                | elif(var_2 == "34"):
                |   movej(p[-0.62575,-0.525,0.05075,2.230,2.215,0])
                | elif(var_2 == "35"):
                |   movej(p[-0.72575,0.525,0.05075,2.230,2.215,0])
                | elif(var_2 == "36"):
                |   movej(p[-0.72575,0.350,0.05075,2.230,2.215,0])
                | elif(var_2 == "37"):
                |   movej(p[-0.72575,0.175,0.05075,2.230,2.215,0])
                | elif(var_2 == "38"):
                |   movej(p[-0.72575,0,0.05075,2.230,2.215,0])
                | elif(var_2 == "39"):
                |   movej(p[-0.72575,-0.175,0.05075,2.230,2.215,0])
                | elif(var_2 == "40"):
                |   movej(p[-0.72575,-0.350,0.05075,2.230,2.215,0])
                | elif(var_2 == "41"):
                |   movej(p[-0.72575,-0.525,0.05075,2.230,2.215,0])
                | elif(var_2 == "42"):
                |   movej(p[-0.82575,0.525,0.05075,2.230,2.215,0])
                | elif(var_2 == "43"):
                |   movej(p[-0.82575,0.350,0.05075,2.230,2.215,0])
                | elif(var_2 == "44"):
                |   movej(p[-0.82575,0.175,0.05075,2.230,2.215,0])
                | elif(var_2 == "45"):
                |   movej(p[-0.82575,0,0.05075,2.230,2.215,0])
                | elif(var_2 == "46"):
                |   movej(p[-0.82575,-0.175,0.05075,2.230,2.215,0])
                | elif(var_2 == "47"):
                |   movej(p[-0.82575,-0.350,0.05075,2.230,2.215,0])
                | elif(var_2 == "48"):
                |   movej(p[-0.82575,-0.525,0.05075,2.230,2.215,0])
                | elif(var_2 == "49"):
                |   movej(p[-0.92575,0.525,0.05075,2.230,2.215,0])
                | elif(var_2 == "50"):
                |   movej(p[-0.92575,0.350,0.05075,2.230,2.215,0])
                | elif(var_2 == "51"):
                |   movej(p[-0.92575,0.175,0.05075,2.230,2.215,0])
                | elif(var_2 == "52"):
                |   movej(p[-0.92575,0,0.05075,2.230,2.215,0])
                | elif(var_2 == "53"):
                |   movej(p[-0.92575,-0.175,0.05075,2.230,2.215,0])
                | elif(var_2 == "54"):
                |   movej(p[-0.92575,-0.350,0.05075,2.230,2.215,0])
                | elif(var_2 == "55"):
                |   movej(p[-0.92575,-0.525,0.05075,2.230,2.215,0])
                | elif(var_2 == "56"):
                |   movej(p[-1.02575,0.525,0.05075,2.230,2.215,0])
                | elif(var_2 == "57"):
                |   movej(p[-1.02575,0.350,0.05075,2.230,2.215,0])
                | elif(var_2 == "58"):
                |   movej(p[-1.02575,0.175,0.05075,2.230,2.215,0])
                | elif(var_2 == "59"):
                |   movej(p[-1.02575,0,0.05075,2.230,2.215,0])
                | elif(var_2 == "60"):
                |   movej(p[-1.02575,-0.175,0.05075,2.230,2.215,0])
                | elif(var_2 == "61"):
                |   movej(p[-1.02575,-0.350,0.05075,2.230,2.215,0])
                | elif(var_2 == "62"):
                |   movej(p[-1.02575,-0.525,0.05075,2.230,2.215,0])
                | elif(var_2 == "71"):
                |   movej(p[-0.600,-1.050,-0.220,0,3.14,0])
                | elif(var_2 == "72"):
                |   movej(p[-0.380,-1.050,-0.220,0,3.14,0])
                | elif(var_2 == "73"):
                |   movej(p[-0.160,-1.050,-0.220,0,3.14,0])
                | elif(var_2 == "74"):
                |   movej(p[0.060,-1.050,-0.220,0,3.14,0])
                | elif(var_2 == "75"):
                |   movej(p[0.280,-1.050,-0.220,0,3.14,0])
                | elif(var_2 == "76"):
                |   movej(p[0.500,-1.050,-0.220,0,3.14,0])
                | end
              Wait Sleep waitTime=0.5
              top_pos1 := get_actual_tcp_pose()
              Script: top_pos1[2] = top_pos1[2]-0.15
              MoveJ speed 60 deg/s, acceleration 80 deg/s^2 (useActiveTCP=true)
                Waypoint Waypoint (Variable): variable=top_pos1
              URCap Vacuum (Robotiq_Grippers, Robotiq Inc.) dataModel(Vacuum.Command.Action=1, Vacuum.Command.PumpAutoCloseDelayInMilliseconds=3000, Vacuum.Command.ShutOffDistance=5.0)
              Wait Sleep waitTime=0.5
              Script: var_4 =  False
              MoveJ speed 60 deg/s, acceleration 80 deg/s^2 (useActiveTCP=true)
                Waypoint place_pos: motionParameters(blendRadius=0.05); TCP in base x=-418.268 y=159.557 z=391.133 mm, rx=-2.2681 ry=-2.171 rz=-0.0004 rad; joints [-180.311, -63.896, -116.331, -89.8, 89.467, 2.625] deg; flange x=-418.043 y=159.256 z=582.133 mm, rx=-2.2681 ry=-2.171 rz=-0.0004 rad
            Else 
              MoveJ speed 60 deg/s, acceleration 80 deg/s^2 (useActiveTCP=true)
                Waypoint place_pos: motionParameters(blendRadius=0.05); TCP in base x=-418.268 y=159.557 z=391.133 mm, rx=-2.2681 ry=-2.171 rz=-0.0004 rad; joints [-180.311, -63.896, -116.331, -89.8, 89.467, 2.625] deg; flange x=-418.043 y=159.256 z=582.133 mm, rx=-2.2681 ry=-2.171 rz=-0.0004 rad
          Wait Sleep waitTime=0.5
          MoveJ speed 60 deg/s, acceleration 80 deg/s^2 (useActiveTCP=true)
            Waypoint Waypoint_10: TCP in base x=-0.074 y=-449.982 z=400.013 mm, rx=2.1808 ry=-2.261 rz=0.0021 rad; joints [-69.631, -64.171, -115.295, -90.553, 89.57, -67.123] deg; flange x=-0.215 y=-449.768 z=591.013 mm, rx=2.1808 ry=-2.261 rz=0.0021 rad
          Folder T12
            If var_3 =="201"
              MoveJ speed 60 deg/s, acceleration 80 deg/s^2 (useActiveTCP=true)
                Waypoint Waypoint_7: TCP in base x=69.993 y=-340.039 z=51.5 mm, rx=2.1806 ry=-2.2612 rz=0.0018 rad; joints [-50.861, -64.539, -152.673, -52.818, 89.717, -48.758] deg; flange x=69.876 y=-339.852 z=242.5 mm, rx=2.1806 ry=-2.2612 rz=0.0018 rad
              Script: var_4 =  True
            ElseIf var_3 == "202"
              MoveJ speed 60 deg/s, acceleration 80 deg/s^2 (useActiveTCP=true)
                Waypoint Waypoint_8: TCP in base x=-65.595 y=-340.045 z=51.514 mm, rx=2.1805 ry=-2.2613 rz=0.0019 rad; joints [-73.362, -64.391, -152.734, -52.902, 89.747, -71.257] deg; flange x=-65.727 y=-339.849 z=242.514 mm, rx=2.1805 ry=-2.2613 rz=0.0019 rad
              Script: var_4 =  True
            ElseIf var_3 =="203"
              MoveJ speed 60 deg/s, acceleration 80 deg/s^2 (useActiveTCP=true)
                Waypoint Waypoint_9: TCP in base x=-194.737 y=-340.099 z=51.532 mm, rx=2.1807 ry=-2.2612 rz=0.0019 rad; joints [-95.738, -71.977, -149.014, -49.049, 89.723, -93.648] deg; flange x=-194.869 y=-339.905 z=242.532 mm, rx=2.1807 ry=-2.2612 rz=0.0019 rad
              Script: var_4 =  True
            ElseIf var_3 == "204"
              Script: var_4 =  False
            If var_4 ==  True
              URCap Find Surface (Robotiq_Copilot, Robotiq Inc.) dataModel(NodeInitializedKey=true, WaitForSteadyWrenchOptionKey=false, ls_force=10.0, ZeroSensorBeforeKey=true, ls_distance=500.0, ls_speed=50.0, ls_direction=Z-, FindSurfaceFeatureKey=0, ls_if_distance=false, ls_if_force=false); state(isChildrenLocked=true)
                'Add Stop conditions from the Find Surface node'
              URCap Vacuum (Robotiq_Grippers, Robotiq Inc.) dataModel(Vacuum.Command.GripMode=Manual, Vacuum.Command.MinVacuumInPercent=70.0, Vacuum.Command.MaxVacuumInPercent=90.0, Vacuum.Command.Action=0, Vacuum.Command.PumpAutoCloseDelayInMilliseconds=3000, Vacuum.Command.ShutOffDistance=5.0)
              Wait Sleep waitTime=0.5
              top_pos2 := get_actual_tcp_pose()
              Script: top_pos2[2] = top_pos2[2]+0.01
              MoveJ speed 60 deg/s, acceleration 80 deg/s^2 (useActiveTCP=true)
                Waypoint Waypoint (Variable): variable=top_pos2
                Waypoint Waypoint_10: TCP in base x=-0.074 y=-449.982 z=400.013 mm, rx=2.1808 ry=-2.261 rz=0.0021 rad; joints [-69.631, -64.171, -115.295, -90.553, 89.57, -67.123] deg; flange x=-0.215 y=-449.768 z=591.013 mm, rx=2.1808 ry=-2.261 rz=0.0021 rad
              Wait Sleep waitTime=0.5
              MoveJ speed 60 deg/s, acceleration 80 deg/s^2 (useActiveTCP=true)
                Waypoint place_pos: motionParameters(blendRadius=0.05); TCP in base x=-418.268 y=159.557 z=391.133 mm, rx=-2.2681 ry=-2.171 rz=-0.0004 rad; joints [-180.311, -63.896, -116.331, -89.8, 89.467, 2.625] deg; flange x=-418.043 y=159.256 z=582.133 mm, rx=-2.2681 ry=-2.171 rz=-0.0004 rad
              Wait Sleep waitTime=0.5
              Script file /programs/new dir/place3.script
                | (same text as the earlier copy of this file)
              Wait Sleep waitTime=0.5
              top_pos1 := get_actual_tcp_pose()
              Script: top_pos1[2] = top_pos1[2]-0.15
              MoveJ speed 60 deg/s, acceleration 80 deg/s^2 (useActiveTCP=true)
                Waypoint Waypoint (Variable): variable=top_pos1
              URCap Vacuum (Robotiq_Grippers, Robotiq Inc.) dataModel(Vacuum.Command.Action=1, Vacuum.Command.PumpAutoCloseDelayInMilliseconds=3000, Vacuum.Command.ShutOffDistance=5.0)
              Wait Sleep waitTime=0.5
              Script: var_4 =  False
              MoveJ speed 60 deg/s, acceleration 80 deg/s^2 (useActiveTCP=true)
                Waypoint place_pos: motionParameters(blendRadius=0.05); TCP in base x=-418.268 y=159.557 z=391.133 mm, rx=-2.2681 ry=-2.171 rz=-0.0004 rad; joints [-180.311, -63.896, -116.331, -89.8, 89.467, 2.625] deg; flange x=-418.043 y=159.256 z=582.133 mm, rx=-2.2681 ry=-2.171 rz=-0.0004 rad
            Else 
              MoveJ speed 60 deg/s, acceleration 80 deg/s^2 (useActiveTCP=true)
                Waypoint place_pos: motionParameters(blendRadius=0.05); TCP in base x=-418.268 y=159.557 z=391.133 mm, rx=-2.2681 ry=-2.171 rz=-0.0004 rad; joints [-180.311, -63.896, -116.331, -89.8, 89.467, 2.625] deg; flange x=-418.043 y=159.256 z=582.133 mm, rx=-2.2681 ry=-2.171 rz=-0.0004 rad
          MoveJ speed 60 deg/s, acceleration 80 deg/s^2 (useActiveTCP=true)
            Waypoint Waypoint_10: TCP in base x=-0.074 y=-449.982 z=400.013 mm, rx=2.1808 ry=-2.261 rz=0.0021 rad; joints [-69.631, -64.171, -115.295, -90.553, 89.57, -67.123] deg; flange x=-0.215 y=-449.768 z=591.013 mm, rx=2.1808 ry=-2.261 rz=0.0021 rad
          Script: socket_send_string("top_placed")
          Wait Sleep waitTime=0.5
          If var_2 == "5"
            MoveJ speed 60 deg/s, acceleration 80 deg/s^2 (useActiveTCP=true)
              Waypoint place_pos: motionParameters(blendRadius=0.05); TCP in base x=-418.268 y=159.557 z=391.133 mm, rx=-2.2681 ry=-2.171 rz=-0.0004 rad; joints [-180.311, -63.896, -116.331, -89.8, 89.467, 2.625] deg; flange x=-418.043 y=159.256 z=582.133 mm, rx=-2.2681 ry=-2.171 rz=-0.0004 rad
            Script: break
      Folder Push
        var_5 := 0
        Wait Sleep waitTime=0.5
        If var_5 == 0
          MoveJ speed 60 deg/s, acceleration 80 deg/s^2 (useActiveTCP=true)
            Waypoint Waypoint_12: TCP in base x=-158.301 y=504.125 z=400.028 mm, rx=-0.0124 ry=-3.1401 rz=0.0022 rad; joints [-235.391, -72.645, -110.118, -87.346, 89.583, -144.51] deg; flange x=-158.011 y=504.388 z=591.028 mm, rx=-0.0124 ry=-3.1401 rz=0.0022 rad
            Waypoint Waypoint_15: TCP in base x=-170.086 y=486.92 z=61.096 mm, rx=-0.0304 ry=-3.1398 rz=0.0019 rad; joints [-232.86, -86.331, -137.199, -46.56, 89.659, -141.738] deg; flange x=-169.765 y=487.153 z=252.096 mm, rx=-0.0304 ry=-3.1398 rz=0.0019 rad
          Wait Sleep waitTime=0.5
          MoveL speed 250 mm/s, acceleration 1200 mm/s^2 (useActiveTCP=true) feature=Base
            Waypoint Waypoint_13: TCP in base x=-1165 y=500.206 z=60.955 mm, rx=-0.0455 ry=-3.1398 rz=0.002 rad; joints [-195.929, -158.624, -21.708, -89.701, 88.788, -104.245] deg; flange x=-1164.721 y=500.444 z=251.955 mm, rx=-0.0455 ry=-3.1398 rz=0.002 rad
          Wait Sleep waitTime=0.5
          Script: var_5 = var_5 + 1
          Script: var_2 = "1"
        Loop Forever
          Script file /programs/new dir/place4.script
            | if(var_2 == "0"):
            |   movej(p[-0.52,0.5,0.15075,2.22,2.22,0])
            | elif(var_2 == "1"):
            |   movej(p[-0.52,0.3,0.15075,2.22,2.22,0])
            | elif(var_2 == "2"):
            |   movej(p[-0.52,0.1,0.15075,2.22,2.22,0])
            | elif(var_2 == "3"):
            |   movej(p[-0.52,-0.1,0.15075,2.22,2.22,0])
            | elif(var_2 == "4"):
            |   movej(p[-0.52,-0.3,0.15075,2.22,2.22,0])
            | elif(var_2 == "5"):
            |   movej(p[-0.52,-0.5,0.15075,2.22,2.22,0])
            | elif(var_2 == "6"):
            |   movej(p[-0.22575,-0.525,0.05075,2.230,2.215,0])
            | elif(var_2 == "7"):
            |   movej(p[-0.32575,0.525,0.05075,2.230,2.215,0])
            | elif(var_2 == "8"):
            |   movej(p[-0.32575,0.350,0.05075,2.230,2.215,0])
            | elif(var_2 == "9"):
            |   movej(p[-0.32575,0.175,0.05075,2.230,2.215,0])
            | elif(var_2 == "10"):
            |   movej(p[-0.32575,0,0.05075,2.230,2.215,0])
            | elif(var_2 == "11"):
            |   movej(p[-0.32575,-0.175,0.05075,2.230,2.215,0])
            | elif(var_2 == "12"):
            |   movej(p[-0.32575,-0.350,0.05075,2.230,2.215,0])
            | elif(var_2 == "13"):
            |   movej(p[-0.32575,-0.525,0.05075,2.230,2.215,0])
            | elif(var_2 == "14"):
            |   movej(p[-0.42575,0.525,0.05075,2.230,2.215,0])
            | elif(var_2 == "15"):
            |   movej(p[-0.42575,0.350,0.05075,2.230,2.215,0])
            | elif(var_2 == "16"):
            |   movej(p[-0.42575,0.175,0.05075,2.230,2.215,0])
            | elif(var_2 == "17"):
            |   movej(p[-0.42575,0,0.05075,2.230,2.215,0])
            | elif(var_2 == "18"):
            |   movej(p[-0.42575,-0.175,0.05075,2.230,2.215,0])
            | elif(var_2 == "19"):
            |   movej(p[-0.42575,-0.350,0.05075,2.230,2.215,0])
            | elif(var_2 == "20"):
            |   movej(p[-0.42575,-0.525,0.05075,2.230,2.215,0])
            | elif(var_2 == "21"):
            |   movej(p[-0.52575,0.525,0.05075,2.230,2.215,0])
            | elif(var_2 == "22"):
            |   movej(p[-0.52575,0.350,0.05075,2.230,2.215,0])
            | elif(var_2 == "23"):
            |   movej(p[-0.52575,0.175,0.05075,2.230,2.215,0])
            | elif(var_2 == "24"):
            |   movej(p[-0.52575,0,0.05075,2.230,2.215,0])
            | elif(var_2 == "25"):
            |   movej(p[-0.52575,-0.175,0.05075,2.230,2.215,0])
            | elif(var_2 == "26"):
            |   movej(p[-0.52575,-0.350,0.05075,2.230,2.215,0])
            | elif(var_2 == "27"):
            |   movej(p[-0.52575,-0.525,0.05075,2.230,2.215,0])
            | elif(var_2 == "28"):
            |   movej(p[-0.62575,0.525,0.05075,2.230,2.215,0])
            | elif(var_2 == "29"):
            |   movej(p[-0.62575,0.350,0.05075,2.230,2.215,0])
            | elif(var_2 == "30"):
            |   movej(p[-0.62575,0.175,0.05075,2.230,2.215,0])
            | elif(var_2 == "31"):
            |   movej(p[-0.62575,0,0.05075,2.230,2.215,0])
            | elif(var_2 == "32"):
            |   movej(p[-0.62575,-0.175,0.05075,2.230,2.215,0])
            | elif(var_2 == "33"):
            |   movej(p[-0.62575,-0.350,0.05075,2.230,2.215,0])
            | elif(var_2 == "34"):
            |   movej(p[-0.62575,-0.525,0.05075,2.230,2.215,0])
            | elif(var_2 == "35"):
            |   movej(p[-0.72575,0.525,0.05075,2.230,2.215,0])
            | elif(var_2 == "36"):
            |   movej(p[-0.72575,0.350,0.05075,2.230,2.215,0])
            | elif(var_2 == "37"):
            |   movej(p[-0.72575,0.175,0.05075,2.230,2.215,0])
            | elif(var_2 == "38"):
            |   movej(p[-0.72575,0,0.05075,2.230,2.215,0])
            | elif(var_2 == "39"):
            |   movej(p[-0.72575,-0.175,0.05075,2.230,2.215,0])
            | elif(var_2 == "40"):
            |   movej(p[-0.72575,-0.350,0.05075,2.230,2.215,0])
            | elif(var_2 == "41"):
            |   movej(p[-0.72575,-0.525,0.05075,2.230,2.215,0])
            | elif(var_2 == "42"):
            |   movej(p[-0.82575,0.525,0.05075,2.230,2.215,0])
            | elif(var_2 == "43"):
            |   movej(p[-0.82575,0.350,0.05075,2.230,2.215,0])
            | elif(var_2 == "44"):
            |   movej(p[-0.82575,0.175,0.05075,2.230,2.215,0])
            | elif(var_2 == "45"):
            |   movej(p[-0.82575,0,0.05075,2.230,2.215,0])
            | elif(var_2 == "46"):
            |   movej(p[-0.82575,-0.175,0.05075,2.230,2.215,0])
            | elif(var_2 == "47"):
            |   movej(p[-0.82575,-0.350,0.05075,2.230,2.215,0])
            | elif(var_2 == "48"):
            |   movej(p[-0.82575,-0.525,0.05075,2.230,2.215,0])
            | elif(var_2 == "49"):
            |   movej(p[-0.92575,0.525,0.05075,2.230,2.215,0])
            | elif(var_2 == "50"):
            |   movej(p[-0.92575,0.350,0.05075,2.230,2.215,0])
            | elif(var_2 == "51"):
            |   movej(p[-0.92575,0.175,0.05075,2.230,2.215,0])
            | elif(var_2 == "52"):
            |   movej(p[-0.92575,0,0.05075,2.230,2.215,0])
            | elif(var_2 == "53"):
            |   movej(p[-0.92575,-0.175,0.05075,2.230,2.215,0])
            | elif(var_2 == "54"):
            |   movej(p[-0.92575,-0.350,0.05075,2.230,2.215,0])
            | elif(var_2 == "55"):
            |   movej(p[-0.92575,-0.525,0.05075,2.230,2.215,0])
            | elif(var_2 == "56"):
            |   movej(p[-1.02575,0.525,0.05075,2.230,2.215,0])
            | elif(var_2 == "57"):
            |   movej(p[-1.02575,0.350,0.05075,2.230,2.215,0])
            | elif(var_2 == "58"):
            |   movej(p[-1.02575,0.175,0.05075,2.230,2.215,0])
            | elif(var_2 == "59"):
            |   movej(p[-1.02575,0,0.05075,2.230,2.215,0])
            | elif(var_2 == "60"):
            |   movej(p[-1.02575,-0.175,0.05075,2.230,2.215,0])
            | elif(var_2 == "61"):
            |   movej(p[-1.02575,-0.350,0.05075,2.230,2.215,0])
            | elif(var_2 == "62"):
            |   movej(p[-1.02575,-0.525,0.05075,2.230,2.215,0])
            | elif(var_2 == "71"):
            |   movej(p[-0.600,-1.050,-0.220,0,3.14,0])
            | elif(var_2 == "72"):
            |   movej(p[-0.380,-1.050,-0.220,0,3.14,0])
            | elif(var_2 == "73"):
            |   movej(p[-0.160,-1.050,-0.220,0,3.14,0])
            | elif(var_2 == "74"):
            |   movej(p[0.060,-1.050,-0.220,0,3.14,0])
            | elif(var_2 == "75"):
            |   movej(p[0.280,-1.050,-0.220,0,3.14,0])
            | elif(var_2 == "76"):
            |   movej(p[0.500,-1.050,-0.220,0,3.14,0])
            | end
          top_pos1 := get_actual_tcp_pose()
          Script: top_pos1[2] = top_pos1[2]-0.085
          Script: top_pos1[0] = top_pos1[0]+0.075
          MoveJ speed 60 deg/s, acceleration 80 deg/s^2 (useActiveTCP=true)
            Waypoint Waypoint (Variable): variable=top_pos1
          Wait Sleep waitTime=0.5
          MoveL speed 250 mm/s, acceleration 1200 mm/s^2 (useActiveTCP=true) feature=Base
            Waypoint Waypoint_14: TCP in base x=-445.061 y=560.023 z=65.015 mm, rx=2.2206 ry=2.2208 rz=-0.0015 rad; joints [-218.809, -104.036, -116.563, -49.549, 89.379, -38.808] deg; flange x=-445.077 y=560.297 z=256.015 mm, rx=2.2206 ry=2.2208 rz=-0.0015 rad
          top_pos3 := get_actual_tcp_pose()
          Script: top_pos3[2] = top_pos1[2]+0.1
          Wait Sleep waitTime=0.5
          MoveJ speed 60 deg/s, acceleration 80 deg/s^2 (useActiveTCP=true)
            Waypoint Waypoint (Variable): variable=top_pos3
            Waypoint place_pos: motionParameters(blendRadius=0.05); TCP in base x=-418.268 y=159.557 z=391.133 mm, rx=-2.2681 ry=-2.171 rz=-0.0004 rad; joints [-180.311, -63.896, -116.331, -89.8, 89.467, 2.625] deg; flange x=-418.043 y=159.256 z=582.133 mm, rx=-2.2681 ry=-2.171 rz=-0.0004 rad
          Wait Sleep waitTime=0.5
          MoveJ speed 60 deg/s, acceleration 80 deg/s^2 (useActiveTCP=true)
            Waypoint Waypoint_12: TCP in base x=-158.301 y=504.125 z=400.028 mm, rx=-0.0124 ry=-3.1401 rz=0.0022 rad; joints [-235.391, -72.645, -110.118, -87.346, 89.583, -144.51] deg; flange x=-158.011 y=504.388 z=591.028 mm, rx=-0.0124 ry=-3.1401 rz=0.0022 rad
            Waypoint Waypoint_15: TCP in base x=-170.086 y=486.92 z=61.096 mm, rx=-0.0304 ry=-3.1398 rz=0.0019 rad; joints [-232.86, -86.331, -137.199, -46.56, 89.659, -141.738] deg; flange x=-169.765 y=487.153 z=252.096 mm, rx=-0.0304 ry=-3.1398 rz=0.0019 rad
          Wait Sleep waitTime=0.5
          MoveL speed 250 mm/s, acceleration 1200 mm/s^2 (useActiveTCP=true) feature=Base
            Waypoint Waypoint_13: TCP in base x=-1165 y=500.206 z=60.955 mm, rx=-0.0455 ry=-3.1398 rz=0.002 rad; joints [-195.929, -158.624, -21.708, -89.701, 88.788, -104.245] deg; flange x=-1164.721 y=500.444 z=251.955 mm, rx=-0.0455 ry=-3.1398 rz=0.002 rad
          Wait Sleep waitTime=0.5
          MoveJ speed 60 deg/s, acceleration 80 deg/s^2 (useActiveTCP=true)
            Waypoint place_pos: motionParameters(blendRadius=0.05); TCP in base x=-418.268 y=159.557 z=391.133 mm, rx=-2.2681 ry=-2.171 rz=-0.0004 rad; joints [-180.311, -63.896, -116.331, -89.8, 89.467, 2.625] deg; flange x=-418.043 y=159.256 z=582.133 mm, rx=-2.2681 ry=-2.171 rz=-0.0004 rad
          Wait Sleep waitTime=0.5
          If var_5 == 1
            Script: var_2 = "2"
            Script: var_5 = var_5 + 1
          ElseIf var_5 == 2
            Script: var_2 = "3"
            Script: var_5 = var_5 + 1
          ElseIf var_5 == 3
            Script: var_2 = "4"
            Script: var_5 = var_5 + 1
          ElseIf var_5 == 4
            Script: var_2 = "5"
            Script: var_5 = var_5 + 1
          ElseIf var_5 == 5
            Script: break
      MoveJ speed 60 deg/s, acceleration 80 deg/s^2 (useActiveTCP=true)
        Waypoint place_pos: motionParameters(blendRadius=0.05); TCP in base x=-418.268 y=159.557 z=391.133 mm, rx=-2.2681 ry=-2.171 rz=-0.0004 rad; joints [-180.311, -63.896, -116.331, -89.8, 89.467, 2.625] deg; flange x=-418.043 y=159.256 z=582.133 mm, rx=-2.2681 ry=-2.171 rz=-0.0004 rad
      MoveJ speed 60 deg/s, acceleration 80 deg/s^2 (useActiveTCP=true)
        Waypoint pick_pos: TCP in base x=419.429 y=-156.467 z=391.085 mm, rx=2.1805 ry=-2.2613 rz=0.0028 rad; joints [0.107, -63.9, -116.333, -89.801, 89.474, 2.62] deg; flange x=419.222 y=-156.192 z=582.085 mm, rx=2.1805 ry=-2.2613 rz=0.0028 rad
      Popup Message (haltProgram=false message=Program finished inputType=Text)
